// TIA Portal V17 export
// export: Created 2022-10-18T12:02:26.1278761Z, ExportSetting WithDefaults, DisplayName Totally Integrated Automation Portal, DisplayVersion V17, DisplayName TIA Portal Openness, DisplayVersion V17, DisplayName TIA Portal Version Control Interface, DisplayVersion V17, DisplayName TIA Portal Test Suite Advanced, DisplayVersion V17, DisplayName STEP 7 Professional, DisplayVersion V17, DisplayName STEP 7 Safety, DisplayVersion V17, DisplayName WinCC Advanced / Unified PC, DisplayVersion V17
FUNCTION_BLOCK "Block_2_FBD"   // FB2, FBD
{ S7_Optimized_Access := 'TRUE' }
VERSION : 0.1
// stored: AutoNumber true, IsIECCheckEnabled false, IsRetainMemResEnabled false, MemoryReserve 100, SetENOAutomatically false, UDAEnableTagReadback false
   VAR
      nCounter2 : Int;
      Trigger : F_TRIG;
   END_VAR
   VAR RETAIN
      IEC_Counter_0_Instance { S7_SetPoint := 'True'} : CTU_INT;
   END_VAR
   VAR CONSTANT
      CounterReset : Int := 50;
   END_VAR
BEGIN

REGION Network 1
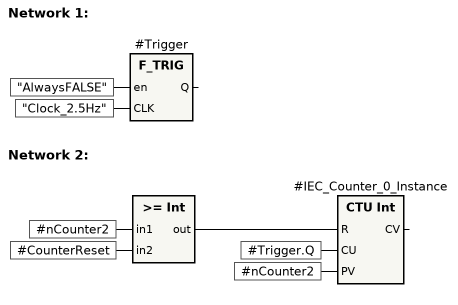
   IF "AlwaysFALSE" THEN
       #Trigger(CLK := "Clock_2.5Hz");   // F_TRIG
   END_IF;
END_REGION

REGION Network 2
   #IEC_Counter_0_Instance(R := #nCounter2 >= #CounterReset, CU := #Trigger.Q, PV := #nCounter2);   // CTU
END_REGION
END_FUNCTION_BLOCK
